{attribute 'linkalways'} 
{attribute 'no_explicit_call' := 'This FB is a CLASS and must be accessed using methods or properties'}
{attribute 'enable_dynamic_creation'}
FUNCTION_BLOCK Node_F_VN_GetAt_TcVnVector3_UINT EXTENDS VisionNode
VAR
    ipContainer : _ITcVnContainer;
    aElement : _TcVnVector3_UINT;
    nIndex : _ULINT(0);
    hrPrev : _HRESULT(S_OK);
    hresult : _HRESULT(S_OK);
END_VAR

METHOD PUBLIC  Clone : I_Node
VAR
	pNode : POINTER TO Node_F_VN_GetAt_TcVnVector3_UINT;
END_VAR
pNode := __NEW(Node_F_VN_GetAt_TcVnVector3_UINT);
Clone := pNode^;
END_METHOD

METHOD FB_init : BOOL
VAR_INPUT
	bInitRetains : BOOL; // if TRUE, the retain variables are initialized (warm start / cold start)
	bInCopyCode : BOOL;  // if TRUE, the instance afterwards gets moved into the copy code (online change)
END_VAR
AddInput('ipContainer', ipContainer);
AddInput('nIndex', nIndex);
AddInput('hrPrev', hrPrev);
AddOutput('aElement', aElement);
AddOutput('hresult',hresult);
END_METHOD

METHOD PROTECTED OnExecute : HRESULT
hresult.Value := F_VN_GetAt_TcVnVector3_UINT(
    ipContainer := ipContainer.Value,
    aElement := aElement.Value,
    nIndex := nIndex.Value,
    hrPrev:= hrPrev.Value);
END_METHOD

METHOD PUBLIC PreExecutionCheck
VAR_INPUT
	Check : I_PreExecutionChecks;
END_VAR
Check.IsTrue(ipContainer.IsValid, 'ipContainer must be a valid container');
Check.IsTrue(ipContainer.HasType(TC_GLOBAL_CONST_LIST.ContainerType_Vector_TcVnVector3_UINT), 'ipContainer contains incorrect type');
END_METHOD

END_FUNCTION_BLOCK

(* stored: Version 1.1.0.1, ProductVersion 3.1.4024.13
   POU Node_F_VN_GetAt_TcVnVector3_UINT: Id {a7baee7a-39b8-482a-b52a-fd41a4eda2ab}, SpecialFunc None
   Folder Constructor: Id {38a7247a-1d53-46a7-b9af-a55c989684b2}
   Method Clone: Id {fecbffa1-8e6d-4ea6-b9c4-5c144a5ff9e9}
   Method FB_init: Id {2ac68d28-4e35-41f4-aa22-02e91282ca69}
   Method OnExecute: Id {9fac6c5f-c2f1-47ef-80a7-d781d9d1e497}
   Method PreExecutionCheck: Id {b7bf0ded-e59b-4e49-a855-b193d252d20a} *)
